Fanuc KAREL source: ko00065.KL

-- PROVISIONAL review KL for V1013-1; original PC SHA256 c1016ca116af958e65746d59c4bcf98443435588442d9cda401cc1d79c876766
-- Incomplete behavior may be omitted. Consult companion uncertainty JSON. Do not deploy.
PROGRAM KO00065
%NOLOCKGROUP
BEGIN
  -- UNRESOLVED_PC offsets 5-12; opcodes 9D,23
  -- UNRESOLVED_PC offsets 17-63; opcodes 27,22,1C,22,1C,22,31,7E,4A
  -- UNRESOLVED_PC offsets 68-72; opcodes 7F
END KO00065
